// TIA Portal V17 program export: 1 tag tables, 1 data types, 0 data blocks, 6 code blocks (in call order from the OBs), 0 instance data blocks

VAR_GLOBAL   // PLC tag table "Default tag table"
   Clock_Byte AT %MB0 : Byte;
   Clock_10Hz AT %M0.0 : Bool;
   Clock_5Hz AT %M0.1 : Bool;
   "Clock_2.5Hz" AT %M0.2 : Bool;
   Clock_2Hz AT %M0.3 : Bool;
   "Clock_1.25Hz" AT %M0.4 : Bool;
   Clock_1Hz AT %M0.5 : Bool;
   "Clock_0.625Hz" AT %M0.6 : Bool;
   "Clock_0.5Hz" AT %M0.7 : Bool;
   System_Byte AT %MB1 : Byte;
   FirstScan AT %M1.0 : Bool;
   DiagStatusUpdate AT %M1.1 : Bool;
   AlwaysTRUE AT %M1.2 : Bool;
   AlwaysFALSE AT %M1.3 : Bool;
END_VAR

TYPE "YourRecipeUDT"
   STRUCT
      "bool" : Bool;
      "int" : Int := 100;
      "dint" : DInt := 9876;
      "string" : String := 'a recipe';
   END_STRUCT;
END_TYPE

ORGANIZATION_BLOCK "Main"   // OB1, LAD, ProgramCycle
TITLE = "Main Program Sweep (Cycle)"
{ S7_Optimized_Access := 'TRUE' }
VERSION : 0.1
// stored: AutoNumber true, IsIECCheckEnabled false, SetENOAutomatically false
   VAR_INPUT
      Initial_Call : Bool;   // Initial call of this OB
      Remanence : Bool;   // =True, if remanent data are available
   END_VAR
BEGIN
END_ORGANIZATION_BLOCK

FUNCTION_BLOCK "WZALib_Debouncer"
TITLE = WZALib_Debouncer
{ S7_Optimized_Access := 'TRUE' }
AUTHOR : WZAutomation
VERSION : 0.1
//For more information, contact WZAutomation: contact@wzautomation.com. Use PLC system clock to perform time based boolean signal debounce hence the number of timer used for this purpose is significantly reduced.
   VAR DB_SPECIFIC
      Loc_Time_Raw : Date_And_Time;
      Loc_Time { ExternalAccessible := 'False'; ExternalVisible := 'False'; ExternalWritable := 'False'} AT Loc_Time_Raw : Date_And_Time;
   END_VAR

   VAR_TEMP 
      RD_LOC_T_Ret : Int;
   END_VAR


BEGIN
	(*-----------------------------------------------------------------------------------------------------------------------------------------
	WZAutomationLib
	For more information, contact WZAutomation: contact@wzautomation.com
	
	-----------------------------------------------------------------------------------------------------------------------------------------*)
	#RD_LOC_T_Ret := RD_LOC_T(#Loc_Time_Raw);
END_FUNCTION_BLOCK

FUNCTION_BLOCK "WZALib_OnOffButton"
TITLE = WZALib_On/OffButton
{ S7_Optimized_Access := 'TRUE' }
AUTHOR : WZAutomation
VERSION : 1.0
//(*----------------------------------------------------------------------------------------------------------------------------------------------*
//*WZAutomationLib CopyRight: WZAutomation                                                                                                        *
//*-----------------------------------------------------------------------------------------------------------------------------------------------*
//*For single button input to alternate a boolean.                                                                                                *
//*-----------------------------------------------------------------------------------------------------------------------------------------------*
//*Variables:                                                                                                                                     *
//*InButton: boolean input to alternate                                                                                                           *
//*                                                                                                                                               *
//*OutSwitch: boolean alternating.                                                                                                                *
//*-----------------------------------------------------------------------------------------------------------------------------------------------*
//*For more information, contact WZAutomation: contact@wzautomation.com                                                                           *
//*-----------------------------------------------------------------------------------------------------------------------------------------------*)
   VAR_INPUT 
      InButton : Bool;   // Push button input signal
   END_VAR

   VAR_OUTPUT 
      OutSwitch : Bool;   // Push button on/off state
   END_VAR

   VAR 
      ButtonState : Bool;   // Button state for FB calculation
      InputFTrig {InstructionName := 'F_TRIG'; LibVersion := '1.0'; S7_SetPoint := 'False'} : F_TRIG;   // Detect the input button signals falling edge
   END_VAR


BEGIN
	(*----------------------------------------------------------------------------------------------------------------------------------------------*
	*WZAutomationLib CopyRight: WZAutomation                                                                                                        *
	*-----------------------------------------------------------------------------------------------------------------------------------------------*
	*For single button input to alternate a boolean.                                                                                                *
	*-----------------------------------------------------------------------------------------------------------------------------------------------*
	*Variables:                                                                                                                                     *
	*InButton: boolean input to alternate                                                                                                           *
	*                                                                                                                                               *
	*OutSwitch: boolean alternating.                                                                                                                *
	*-----------------------------------------------------------------------------------------------------------------------------------------------*
	*For more information, contact WZAutomation: contact@wzautomation.com                                                                           *
	*-----------------------------------------------------------------------------------------------------------------------------------------------*)
	REGION Input Falling Edge
	    //Catch the falling edge of the input button signal
	    #InputFTrig(CLK := #InButton);
	END_REGION
	
	REGION Alternate Output
	    //Generate button state based on memory
	    IF #InputFTrig.Q AND #ButtonState THEN
	        #ButtonState := FALSE;
	    ELSIF #InputFTrig.Q AND NOT #ButtonState THEN
	        #ButtonState := TRUE;
	    END_IF;
	    
	    
	    //Output the alternating state
	    #OutSwitch := #ButtonState;
	END_REGION
END_FUNCTION_BLOCK

FUNCTION_BLOCK "WZALib_Ramp"
TITLE = WZALib_Ramp
{ S7_Optimized_Access := 'TRUE' }
AUTHOR : WZAutomation
VERSION : 1.0
//(*----------------------------------------------------------------------------------------------------------------------------------------------*
//*WZAutomationLib CopyRight: WZAutomation                                                                                                        *
//*-----------------------------------------------------------------------------------------------------------------------------------------------*
//*Generate ramp based on input target value, ramp mode and ramp rate or ramp time.                                                               *
//*Rampmode TRUE: the ramp output will be fixed to the ramp time specified in the input. The ramp rate (slope) will be adjusted to the fixed time *
//*and the difference between the ramp start and end values.                                                                                      *
//*Rampmode FALSE: the ramp output will be fixed to the ramp rate and the time for the output to reach the target value varies.                   *
//*This ramp only generates linear ramp with f(x)=kx+b.                                                                                           *
//*-----------------------------------------------------------------------------------------------------------------------------------------------*
//*Variables:                                                                                                                                     *
//*InRampMode: ramp mode, True = Fixed Ramp time, False = Fixed rate.                                                                             *
//*InTargetValue: the value that the ramp should reach at the end of the slope.                                                                   *
//*InRampeRate: the slope of the ramp expression. Unit: value / second.                                                                           *
//*InRampTime: the time (x) of the ramp expression. Unit: ms.                                                                                     *
//*                                                                                                                                               *
//*OutRamping: the ramp is running.                                                                                                               *
//*OutCurrentValue: current value of the ramp.                                                                                                    *
//*OutCurrentRampTime: current time of the ramp.                                                                                                  *
//*-----------------------------------------------------------------------------------------------------------------------------------------------*
//*For more information, contact WZAutomation: contact@wzautomation.com                                                                           *
//*-----------------------------------------------------------------------------------------------------------------------------------------------*)
   VAR_INPUT 
      InRampMode : Bool;   // True = Fixed Ramp time, False = Fixed rate
      InTargetValue : Real;
      InRampRate : Real := 1.0;   // value / second
      InRampTime : Time := T#10ms;
   END_VAR

   VAR_OUTPUT 
      OutRamping : Bool;
      OutCurrentValue : Real;
      OutCurrentRampTime : Time;
   END_VAR

   VAR 
      TargetValueMem : Real;
      CurrentValue : Real;
      StartValue : Real;
      EndValue : Real;
      ValueDiff : Real;
      TimeDiffReal : Real;
      RampRate : Real;
      CurrentTime : Time;
      EndTime : Time;
      RampTimerPT : Time;
      RampTimer_FixedTime {InstructionName := 'TON_TIME'; LibVersion := '1.0'; S7_SetPoint := 'False'} : TON_TIME;
      RampTimer_FixedRate {InstructionName := 'TON_TIME'; LibVersion := '1.0'} : TON_TIME;
   END_VAR


BEGIN
	(*----------------------------------------------------------------------------------------------------------------------------------------------*
	*WZAutomationLib CopyRight: WZAutomation                                                                                                        *
	*-----------------------------------------------------------------------------------------------------------------------------------------------*
	*Generate ramp based on input target value, ramp mode and ramp rate or ramp time.                                                               *
	*Rampmode TRUE: the ramp output will be fixed to the ramp time specified in the input. The ramp rate (slope) will be adjusted to the fixed time *
	*and the difference between the ramp start and end values.                                                                                      *
	*Rampmode FALSE: the ramp output will be fixed to the ramp rate and the time for the output to reach the target value varies.                   *
	*This ramp only generates linear ramp with f(x)=kx+b.                                                                                           *
	*-----------------------------------------------------------------------------------------------------------------------------------------------*
	*Variables:                                                                                                                                     *
	*InRampMode: ramp mode, True = Fixed Ramp time, False = Fixed rate.                                                                             *
	*InTargetValue: the value that the ramp should reach at the end of the slope.                                                                   *
	*InRampeRate: the slope of the ramp expression. Unit: value / second.                                                                           *
	*InRampTime: the time (x) of the ramp expression. Unit: ms.                                                                                     *
	*                                                                                                                                               *
	*OutRamping: the ramp is running.                                                                                                               *
	*OutCurrentValue: current value of the ramp.                                                                                                    *
	*OutCurrentRampTime: current time of the ramp.                                                                                                  *
	*-----------------------------------------------------------------------------------------------------------------------------------------------*
	*For more information, contact WZAutomation: contact@wzautomation.com                                                                           *
	*-----------------------------------------------------------------------------------------------------------------------------------------------*)
	REGION Value Preperation
	    //Update ramp settings upon input value change
	    IF #InTargetValue <> #TargetValueMem THEN
	        #StartValue := #CurrentValue;
	        #TargetValueMem := #EndValue := #InTargetValue;
	        
	        IF #InRampMode THEN
	            //Fixed time ramp settings
	            IF #InRampTime > T#0s THEN
	                #EndTime := #RampTimerPT := #InRampTime;
	                #TimeDiffReal := UDINT_TO_REAL(IN := TIME_TO_UDINT(IN := #InRampTime));
	            ELSE
	                #EndTime := #RampTimerPT := T#10ms;
	                #TimeDiffReal := UDINT_TO_REAL(IN := TIME_TO_UDINT(IN := T#10ms));
	            END_IF;
	            
	            #ValueDiff := #EndValue - #StartValue;
	            #RampRate := #ValueDiff / #TimeDiffReal;
	            RESET_TIMER(#RampTimer_FixedTime);
	            
	        ELSE
	            //Fixed rate ramp settings
	            IF #InRampRate <> 0.0 THEN
	                #RampRate := #InRampRate;
	            ELSE
	                #RampRate := 1000.0;
	            END_IF;
	            
	            #ValueDiff := ABS(IN := #EndValue - #StartValue);
	            #TimeDiffReal := 1000 * #ValueDiff / #RampRate;
	            #EndTime := #RampTimerPT := UDINT_TO_TIME(IN := REAL_TO_UDINT(IN := #TimeDiffReal));
	            
	            IF #EndValue < #StartValue THEN
	                #RampRate := - #RampRate;
	            END_IF;
	            
	            RESET_TIMER(#RampTimer_FixedRate);
	            
	        END_IF;
	        
	    END_IF;
	    
	END_REGION
	
	REGION Ramp Timer
	    //Run ramp timer
	    #RampTimer_FixedTime(IN := (#InRampMode AND #CurrentValue <> #TargetValueMem) OR #RampTimer_FixedTime.Q,
	                         PT := #RampTimerPT);
	    
	    #RampTimer_FixedRate(IN := (NOT #InRampMode AND #CurrentValue <> #TargetValueMem) OR #RampTimer_FixedRate.Q,
	                         PT := #RampTimerPT);
	    
	END_REGION
	
	REGION Ramp Calculation
	    #OutRamping := #RampTimerPT > T#0s AND (#InRampMode AND NOT #RampTimer_FixedTime.Q OR NOT #InRampMode AND NOT #RampTimer_FixedRate.Q);
	    
	    IF NOT #OutRamping THEN
	        #CurrentValue := #TargetValueMem;
	    END_IF;
	    
	    IF #InRampMode AND #OutRamping THEN
	        #CurrentValue := #RampRate * UDINT_TO_REAL(IN := TIME_TO_UDINT(IN := #RampTimer_FixedTime.ET)) + #StartValue;
	    END_IF;
	    
	    IF NOT #InRampMode AND #OutRamping THEN
	        #CurrentValue := #RampRate * UDINT_TO_REAL(IN := TIME_TO_UDINT(IN := #RampTimer_FixedRate.ET)) / 1000 + #StartValue;
	    END_IF;
	    
	END_REGION
	
	REGION Ramp Status Output
	    IF #InRampMode AND NOT #RampTimer_FixedTime.Q THEN
	        #OutCurrentRampTime := #RampTimer_FixedTime.ET;
	    ELSIF NOT #InRampMode AND NOT #RampTimer_FixedRate.Q THEN
	        #OutCurrentRampTime := #RampTimer_FixedRate.ET;
	    ELSE
	        #OutCurrentRampTime := T#0s;
	    END_IF;
	    
	    #OutCurrentValue := #CurrentValue;
	END_REGION
END_FUNCTION_BLOCK

FUNCTION_BLOCK "WZALib_Sequencer"
TITLE = WZALib_Sequencer
{ S7_Optimized_Access := 'TRUE' }
AUTHOR : WZAutomation
VERSION : 1.0
//(*----------------------------------------------------------------------------------------------------------------------------------------------*
//*WZAutomationLib CopyRight: WZAutomation                                                                                                        *
//*-----------------------------------------------------------------------------------------------------------------------------------------------*
//*For sequence control up to 256 steps.                                                                                                          *
//*In a typical machine automation application, it is normal to control a machine in step sequences. SFC is a good choice though the language     *
//*is heavy comparing with others and most of the scenarios SFC's functions are not fully utilized. WZAutomation made this sequencer with years   *
//*of experience in machine automation.                                                                                                           *
//*-----------------------------------------------------------------------------------------------------------------------------------------------*
//*Variables:                                                                                                                                     *
//*InAuto: the sequence will run if this input is true.                                                                                           *
//*InStepMode: the sequence will run in step mode if InAuto is true.                                                                              *
//*InStepCmd: the sequence will only move one step each time when the step's transition condition is fulfilled and this input sees a rising edge. *
//*InInterlock: interlock the step sequence from moving forward if true.                                                                          *
//*InHoldStepTimer: hold step timer so sequence can stay in a step without timeout.                                                               *
//*InReset: reset the sequence to the default step and state                                                                                      *
//*InNextStep: the next step the sequence is commanded to go to.                                                                                  *
//*InDefaultSteop: the default step when sequence is reset.                                                                                       *
//*InStepTimeOut: set the time for sequence timeout.                                                                                              *
//*                                                                                                                                               *
//*OutSequenceTimeOut: true if sequence is timed out in a step.                                                                                   *
//*OutStepRdytoMove: indicate the sequence is ready to move on in step mode.                                                                      *
//*OutCurrentStep: current step number of the sequence.                                                                                           *
//*OutCurrentStepTime: the time the sequence has been in the current step.                                                                        *
//*-----------------------------------------------------------------------------------------------------------------------------------------------*
//*For more information, contact WZAutomation: contact@wzautomation.com                                                                           *
//*-----------------------------------------------------------------------------------------------------------------------------------------------*)
   VAR_INPUT 
      InAuto : Bool;   // Set sequence in auto mode (automatic step forward if conditions are fulfilled)
      InStepMode : Bool;   // Set sequence in step mode
      InStepCmd : Bool;   // Sequence step forward command
      InInterlock : Bool;   // Sequence interlock command
      InHoldStepTimer : Bool;   // Sequence step timer stop command
      InReset : Bool;   // Sequence reset to default step
      InNextStep : Int;   // Next step number according to sequence
      InDefaultStep : Int;   // Default step number when sequence is reset
      InStepTimeOutTime : Time := T#1s;   // Timeout time setting for the current sequence step
   END_VAR

   VAR_OUTPUT 
      OutSequenceTimeOut : Bool;   // True: Sequence is timed out in a step
      OutStepRdytoMove : Bool;   // Indicate the sequence is ready to move on in step mode
      OutCurrentStep : Int;   // Current step number
      OutCurrentStepTime : Time;   // The time the sequence has been in the current step
   END_VAR

   VAR 
      Steps : Array[0..255] of Bool;   // Steps
      CurrentStep : Int;
      StepTimeOutTime : Time;
      StepCmdRTrig {InstructionName := 'R_TRIG'; LibVersion := '1.0'; S7_SetPoint := 'False'} : R_TRIG;
      StepActiveTime {InstructionName := 'TON_TIME'; LibVersion := '1.0'; S7_SetPoint := 'False'} : TON_TIME;   // Timer for current step time
   END_VAR


BEGIN
	(*----------------------------------------------------------------------------------------------------------------------------------------------*
	*WZAutomationLib CopyRight: WZAutomation                                                                                                        *
	*-----------------------------------------------------------------------------------------------------------------------------------------------*
	*For sequence control up to 256 steps.                                                                                                          *
	*In a typical machine automation application, it is normal to control a machine in step sequences. SFC is a good choice though the language     *
	*is heavy comparing with others and most of the scenarios SFC's functions are not fully utilized. WZAutomation made this sequencer with years   *
	*of experience in machine automation.                                                                                                           *
	*-----------------------------------------------------------------------------------------------------------------------------------------------*
	*Variables:                                                                                                                                     *
	*InAuto: the sequence will run if this input is true.                                                                                           *
	*InStepMode: the sequence will run in step mode if InAuto is true.                                                                              *
	*InStepCmd: the sequence will only move one step each time when the step's transition condition is fulfilled and this input sees a rising edge. *
	*InInterlock: interlock the step sequence from moving forward if true.                                                                          *
	*InHoldStepTimer: hold step timer so sequence can stay in a step without timeout.                                                               *
	*InReset: reset the sequence to the default step and state                                                                                      *
	*InNextStep: the next step the sequence is commanded to go to.                                                                                  *
	*InDefaultSteop: the default step when sequence is reset.                                                                                       *
	*InStepTimeOut: set the time for sequence timeout.                                                                                              *
	*                                                                                                                                               *
	*OutSequenceTimeOut: true if sequence is timed out in a step.                                                                                   *
	*OutStepRdytoMove: indicate the sequence is ready to move on in step mode.                                                                      *
	*OutCurrentStep: current step number of the sequence.                                                                                           *
	*OutCurrentStepTime: the time the sequence has been in the current step.                                                                        *
	*-----------------------------------------------------------------------------------------------------------------------------------------------*
	*For more information, contact WZAutomation: contact@wzautomation.com                                                                           *
	*-----------------------------------------------------------------------------------------------------------------------------------------------*)
	
	REGION Reset Sequence
	    IF #InReset THEN
	        //Set all steps to FALSE
	        FILL_BLK(IN    := FALSE,
	                 COUNT := 256,
	                 OUT   => #Steps[0]);
	        
	        //Set the default start step to TRUE
	        #Steps[#InDefaultStep] := TRUE;
	        #CurrentStep := #InDefaultStep;
	        
	        //Reset step active timer
	        RESET_TIMER(#StepActiveTime);
	        
	        //Update current step time active timer
	        #StepTimeOutTime := #InStepTimeOutTime;
	        
	    END_IF;
	    
	END_REGION
	
	REGION Input Value Process
	    #StepCmdRTrig(CLK := #InStepCmd);
	    
	END_REGION
	
	REGION Sequence Control
	    IF #InAuto AND NOT #InReset THEN
	        IF #InStepMode THEN
	            //If in step mode, the sequence is commanded to move to the next step and there is no interlock to stop it, move on to the next step
	            IF #InNextStep <> #CurrentStep AND NOT #InInterlock AND #StepCmdRTrig.Q THEN
	                #CurrentStep := #InNextStep;
	                
	                //Reset step active time and update the step timeout time
	                RESET_TIMER(#StepActiveTime);
	                IF #StepTimeOutTime <> #InStepTimeOutTime THEN
	                    #StepTimeOutTime := #InStepTimeOutTime;
	                END_IF;
	                
	            END_IF;
	            
	        ELSE
	            //If the sequence is commanded to move to the next step and there is no interlock to stop it, move on to the next step
	            IF #InNextStep <> #CurrentStep AND NOT #InInterlock THEN
	                #CurrentStep := #InNextStep;
	                
	                //Reset step active time and update the step timeout time
	                RESET_TIMER(#StepActiveTime);
	                IF #StepTimeOutTime <> #InStepTimeOutTime THEN
	                    #StepTimeOutTime := #InStepTimeOutTime;
	                END_IF;
	                
	            END_IF;
	            
	        END_IF;
	        
	    END_IF;
	    
	END_REGION
	
	REGION Update Step Array
	    FILL_BLK(IN    := FALSE,
	             COUNT := 256,
	             OUT   => #Steps[0]);
	    
	    #Steps[#CurrentStep] := TRUE;
	    
	END_REGION
	
	REGION Step Active Timer
	    #StepActiveTime(IN := #InNextStep = #CurrentStep AND #InDefaultStep <> #CurrentStep AND #InAuto AND NOT #InHoldStepTimer AND NOT #InStepMode AND NOT #InInterlock,
	                    PT := #StepTimeOutTime);
	    
	END_REGION
	
	REGION Update Output
	    #OutSequenceTimeOut := #StepActiveTime.Q;
	    #OutStepRdytoMove := #InAuto AND #InStepMode AND #InNextStep <> #CurrentStep AND NOT #InInterlock;
	    #OutCurrentStep := #CurrentStep;
	    #OutCurrentStepTime := #StepActiveTime.ET;
	    
	END_REGION
END_FUNCTION_BLOCK

FUNCTION_BLOCK "WZALib_WebServerRecipe"
TITLE = WZALib_WebServerRecipe
{ S7_Optimized_Access := 'TRUE' }
AUTHOR : WZAutomation
VERSION : 1.0
//(*----------------------------------------------------------------------------------------------------------------------------------------------*
//*WZAutomationLib CopyRight: WZAutomation                                                                                                        *
//*-----------------------------------------------------------------------------------------------------------------------------------------------*
//*This function block reads and writes user defined recipe data from and to the PLC integrated webserver interface. Save has the priority.       *
//*-----------------------------------------------------------------------------------------------------------------------------------------------*
//*Variables:                                                                                                                                     *
//*InLoadRecipe: command to trigger a load from the webserver.                                                                                    *
//*InSaveRecipe: command to trigger a save to the webserver                                                                                       *
//*                                                                                                                                               *
//*OutRecipeDiff: At lease one recipe value is different between webserver and PLC                                                                *
//*-----------------------------------------------------------------------------------------------------------------------------------------------*
//*For more information, contact WZAutomation: contact@wzautomation.com                                                                           *
//*-----------------------------------------------------------------------------------------------------------------------------------------------*)
   VAR_INPUT 
      InImportRecipe : Bool;   // Load recipe from webserver
      InExportRecipe : Bool;   // Save recipe to webserver
   END_VAR

   VAR_OUTPUT 
      OutRecipeDiff : Bool;   // At lease one recipe value is different between webserver and PLC
      OutWebServerBusy : Bool;   // PLC is reading or writing the webserver .CSV file
   END_VAR

   VAR 
      ExportReqM : Bool;   // Memory bit for save command
      ImportReqM : Bool;   // Memory bit for load command
      RecipeExport {InstructionName := 'RecipeExport'; LibVersion := '1.2'; S7_SetPoint := 'False'} : RecipeExport;
      RecipeImport {InstructionName := 'RecipeImport'; LibVersion := '1.2'; S7_SetPoint := 'False'} : RecipeImport;
      Recipes { S7_SetPoint := 'False'} : Array[0..#NumofRecipes] of "YourRecipeUDT";   // Recipe Values loaded from the webserver
   END_VAR

   VAR CONSTANT 
      NumofRecipes : Int := 10;   // Number of recipes to be processed - change the value before using it
   END_VAR


BEGIN
	(*----------------------------------------------------------------------------------------------------------------------------------------------*
	*WZAutomationLib CopyRight: WZAutomation                                                                                                        *
	*-----------------------------------------------------------------------------------------------------------------------------------------------*
	*This function block reads and writes user defined recipe data from and to the PLC integrated webserver interface. Save has the priority.       *
	*-----------------------------------------------------------------------------------------------------------------------------------------------*
	*Variables:                                                                                                                                     *
	*InLoadRecipe: command to trigger a load from the webserver.                                                                                    *
	*InSaveRecipe: command to trigger a save to the webserver                                                                                       *
	*                                                                                                                                               *
	*OutRecipeDiff: At lease one recipe value is different between webserver and PLC                                                                *
	*-----------------------------------------------------------------------------------------------------------------------------------------------*
	*For more information, contact WZAutomation: contact@wzautomation.com                                                                           *
	*-----------------------------------------------------------------------------------------------------------------------------------------------*)
	
	REGION Recipe Export
	    IF #InExportRecipe AND NOT #ExportReqM THEN
	        #ExportReqM := TRUE;
	        
	    ELSIF #ExportReqM AND #RecipeExport.DONE AND NOT #InExportRecipe THEN
	        #ExportReqM := FALSE;
	        
	    END_IF;
	    
	    #RecipeExport(REQ       := #ExportReqM,
	                  RECIPE_DB := #Recipes);
	    
	END_REGION
	
	REGION Recipe Import
	    IF #InImportRecipe AND NOT #InExportRecipe AND NOT #ImportReqM THEN
	        #ImportReqM := TRUE;
	        
	    ELSIF #ImportReqM AND #RecipeImport.DONE AND NOT #InImportRecipe THEN
	        #ImportReqM := FALSE;
	        
	    END_IF;
	    
	    #RecipeImport(REQ       := #ImportReqM,
	                  RECIPE_DB := #Recipes);
	    
	END_REGION
	
	REGION Webserver Busy
	    #OutWebServerBusy := #RecipeExport.BUSY OR #RecipeImport.BUSY;
	    
	END_REGION
END_FUNCTION_BLOCK
